# EPICS substitutions: iocBoot/iocTest/testISIS.substitutions
file "db/testISIS.template" { pattern
{P, R, PORT, POLLER, INDEX, SLICE}
{omronEIP:, 0:, omronDriver, slowPoller, 1, 9}
{omronEIP:, 1:, omronDriver, slowPoller, 10, 9}
{omronEIP:, 2:, omronDriver, slowPoller, 19, 9}
{omronEIP:, 3:, omronDriver, slowPoller, 28, 9}
{omronEIP:, 4:, omronDriver, slowPoller, 37, 9}
{omronEIP:, 5:, omronDriver, slowPoller, 46, 9}
{omronEIP:, 6:, omronDriver, slowPoller, 55, 9}
{omronEIP:, 7:, omronDriver, slowPoller, 64, 9}
{omronEIP:, 8:, omronDriver, slowPoller, 73, 9}
{omronEIP:, 9:, omronDriver, slowPoller, 82, 9}
{omronEIP:, 10:, omronDriver, slowPoller, 91, 9}
{omronEIP:, 11:, omronDriver, slowPoller, 100, 9}
{omronEIP:, 12:, omronDriver, slowPoller, 109, 9}
{omronEIP:, 13:, omronDriver, slowPoller, 118, 9}
{omronEIP:, 14:, omronDriver, slowPoller, 127, 9}
{omronEIP:, 15:, omronDriver, slowPoller, 136, 9}
{omronEIP:, 16:, omronDriver, slowPoller, 145, 9}
{omronEIP:, 17:, omronDriver, slowPoller, 154, 9}
{omronEIP:, 18:, omronDriver, slowPoller, 163, 9}
{omronEIP:, 19:, omronDriver, slowPoller, 172, 9}
{omronEIP:, 20:, omronDriver, slowPoller, 181, 9}
{omronEIP:, 21:, omronDriver, slowPoller, 190, 9}
{omronEIP:, 22:, omronDriver, slowPoller, 199, 9}
{omronEIP:, 23:, omronDriver, slowPoller, 208, 9}
{omronEIP:, 24:, omronDriver, slowPoller, 217, 9}
{omronEIP:, 25:, omronDriver, slowPoller, 226, 9}
{omronEIP:, 26:, omronDriver, slowPoller, 235, 9}
{omronEIP:, 27:, omronDriver, slowPoller, 244, 9}
{omronEIP:, 28:, omronDriver, slowPoller, 253, 9}
{omronEIP:, 29:, omronDriver, slowPoller, 262, 9}
{omronEIP:, 30:, omronDriver, slowPoller, 271, 9}
{omronEIP:, 31:, omronDriver, slowPoller, 280, 9}
{omronEIP:, 32:, omronDriver, slowPoller, 289, 9}
{omronEIP:, 33:, omronDriver, slowPoller, 298, 9}
{omronEIP:, 34:, omronDriver, slowPoller, 307, 9}
{omronEIP:, 35:, omronDriver, slowPoller, 316, 9}
{omronEIP:, 36:, omronDriver, slowPoller, 325, 9}
{omronEIP:, 37:, omronDriver, slowPoller, 334, 9}
{omronEIP:, 38:, omronDriver, slowPoller, 343, 9}
{omronEIP:, 39:, omronDriver, slowPoller, 352, 9}
{omronEIP:, 40:, omronDriver, slowPoller, 361, 9}
{omronEIP:, 41:, omronDriver, slowPoller, 370, 9}
{omronEIP:, 42:, omronDriver, slowPoller, 379, 9}
{omronEIP:, 43:, omronDriver, slowPoller, 388, 9}
{omronEIP:, 44:, omronDriver, slowPoller, 397, 9}
{omronEIP:, 45:, omronDriver, slowPoller, 406, 9}
{omronEIP:, 46:, omronDriver, slowPoller, 415, 9}
{omronEIP:, 47:, omronDriver, slowPoller, 424, 9}
{omronEIP:, 48:, omronDriver, slowPoller, 433, 9}
{omronEIP:, 49:, omronDriver, slowPoller, 442, 9}
{omronEIP:, 50:, omronDriver, slowPoller, 451, 9}
{omronEIP:, 51:, omronDriver, slowPoller, 460, 9}
{omronEIP:, 52:, omronDriver, slowPoller, 469, 9}
{omronEIP:, 53:, omronDriver, slowPoller, 478, 9}
{omronEIP:, 54:, omronDriver, slowPoller, 487, 9}
{omronEIP:, 55:, omronDriver, slowPoller, 496, 9}
{omronEIP:, 56:, omronDriver, slowPoller, 505, 9}
{omronEIP:, 57:, omronDriver, slowPoller, 514, 9}
{omronEIP:, 58:, omronDriver, slowPoller, 523, 9}
{omronEIP:, 59:, omronDriver, slowPoller, 532, 9}
{omronEIP:, 60:, omronDriver, slowPoller, 541, 9}
{omronEIP:, 61:, omronDriver, slowPoller, 550, 9}
{omronEIP:, 62:, omronDriver, slowPoller, 559, 9}
{omronEIP:, 63:, omronDriver, slowPoller, 568, 9}
{omronEIP:, 64:, omronDriver, slowPoller, 577, 9}
{omronEIP:, 65:, omronDriver, slowPoller, 586, 9}
{omronEIP:, 66:, omronDriver, slowPoller, 595, 9}
{omronEIP:, 67:, omronDriver, slowPoller, 604, 9}
{omronEIP:, 68:, omronDriver, slowPoller, 613, 9}
{omronEIP:, 69:, omronDriver, slowPoller, 622, 9}
{omronEIP:, 70:, omronDriver, slowPoller, 631, 9}
{omronEIP:, 71:, omronDriver, slowPoller, 640, 9}
{omronEIP:, 72:, omronDriver, slowPoller, 649, 9}
{omronEIP:, 73:, omronDriver, slowPoller, 658, 9}
{omronEIP:, 74:, omronDriver, slowPoller, 667, 9}
{omronEIP:, 75:, omronDriver, slowPoller, 676, 9}
{omronEIP:, 76:, omronDriver, slowPoller, 685, 9}
{omronEIP:, 77:, omronDriver, slowPoller, 694, 9}
{omronEIP:, 78:, omronDriver, slowPoller, 703, 9}
{omronEIP:, 79:, omronDriver, slowPoller, 712, 9}
{omronEIP:, 80:, omronDriver, slowPoller, 721, 9}
{omronEIP:, 81:, omronDriver, slowPoller, 730, 9}
{omronEIP:, 82:, omronDriver, slowPoller, 739, 9}
{omronEIP:, 83:, omronDriver, slowPoller, 748, 9}
{omronEIP:, 84:, omronDriver, slowPoller, 757, 9}
{omronEIP:, 85:, omronDriver, slowPoller, 766, 9}
{omronEIP:, 86:, omronDriver, slowPoller, 775, 9}
{omronEIP:, 87:, omronDriver, slowPoller, 784, 9}
{omronEIP:, 88:, omronDriver, slowPoller, 793, 9}
{omronEIP:, 89:, omronDriver, slowPoller, 802, 9}
{omronEIP:, 90:, omronDriver, slowPoller, 811, 9}
{omronEIP:, 91:, omronDriver, slowPoller, 820, 9}
{omronEIP:, 92:, omronDriver, slowPoller, 829, 9}
{omronEIP:, 93:, omronDriver, slowPoller, 838, 9}
{omronEIP:, 94:, omronDriver, slowPoller, 847, 9}
{omronEIP:, 95:, omronDriver, slowPoller, 856, 9}
{omronEIP:, 96:, omronDriver, slowPoller, 865, 9}
{omronEIP:, 97:, omronDriver, slowPoller, 874, 9}
{omronEIP:, 98:, omronDriver, slowPoller, 883, 9}
{omronEIP:, 99:, omronDriver, slowPoller, 892, 9}
{omronEIP:, 100:, omronDriver, slowPoller, 901, 9}
{omronEIP:, 101:, omronDriver, slowPoller, 910, 9}
{omronEIP:, 102:, omronDriver, slowPoller, 919, 9}
{omronEIP:, 103:, omronDriver, slowPoller, 928, 9}
{omronEIP:, 104:, omronDriver, slowPoller, 937, 9}
{omronEIP:, 105:, omronDriver, slowPoller, 946, 9}
{omronEIP:, 106:, omronDriver, slowPoller, 955, 9}
{omronEIP:, 107:, omronDriver, slowPoller, 964, 9}
{omronEIP:, 108:, omronDriver, slowPoller, 973, 9}
{omronEIP:, 109:, omronDriver, slowPoller, 982, 9}
{omronEIP:, 110:, omronDriver, slowPoller, 991, 9}
{omronEIP:, 111:, omronDriver, slowPoller, 1000, 1}
}
